FUNCTION_BLOCK FB_DisplacementSensor
VAR_INPUT
END_VAR
VAR_OUTPUT
END_VAR
VAR
END_VAR

END_FUNCTION_BLOCK

(* stored: Version 1.1.0.1, ProductVersion 3.1.4024.12
   POU FB_DisplacementSensor: Id {7ba37002-a059-4534-9366-2b290f489892}, SpecialFunc None *)
